KUKA KRL data list: sPlanen2.dat

&ACCESS RVO
DEFDAT sPlanen2
;FOLD EXTERNAL DECLARATIONS;%{PE}%MKUKATPBASIS,%CEXT,%VCOMMON,%P
  ;FOLD BASISTECH EXT;%{PE}%MKUKATPBASIS,%CEXT,%VEXT,%P
    EXT  BAS (BAS_COMMAND  :IN,REAL  :IN )
  ;ENDFOLD (BASISTECH EXT)

;ENDFOLD (EXTERNAL DECLARATIONS)
ENDDAT
